// TIA Portal V16 export
// export: Created 2024-09-05T17:40:14.2825962Z, ExportSetting WithDefaults, DisplayName Totally Integrated Automation Portal, DisplayVersion V16 Update 6, DisplayName TIA Portal Version Control Interface, DisplayVersion V16 Update 2, DisplayName TIA Portal Openness, DisplayVersion V16 Update 6, DisplayName STEP 7 Professional, DisplayVersion V16 Update 6, DisplayName STEP 7 Safety, DisplayVersion V16, DisplayName WinCC Advanced, DisplayVersion V16 Update 6
TYPE "UDT_TurnTableStatus"
// stored: IsFailsafeCompliant false
   STRUCT
      Collision : Bool;
      Communication : Bool;
      EnabledForOneScan : Bool;   // Rising edge status
      IndexerInPositionForOneScan : Bool;   // Rising edge status
      CycleStep : UInt;
      CycleRunning : Bool;
      CycleFinished : Bool;
      CycleStopped : Bool;
      DoneCW : Bool;
      DoneCCW : Bool;
      SafetyPosition : Bool;
      BasicPosition : Bool;
   END_STRUCT;
END_TYPE
